TEXTLIST BDList
  0 = 'Disable'
  1 = 'ForceOn'
  2 = 'ForceOff'
   = ''
END_TEXTLIST

(* stored: Version 1.1.0.1, ProductVersion 3.1.4022.12
   TextList BDList: Id {721cb3dc-de37-4f47-b51d-4c3ccfaebfe8} *)
